TYPE T_Ctrl_SIf_DPJ_Out :
STRUCT
	///switch valve retract
	bolRetract: T_Ctrl_IoBool;
	///switch valve extend
	bolExtend: T_Ctrl_IoBool;
END_STRUCT
END_TYPE

(* stored: Version 1.1.0.1, ProductVersion 3.1.0.19
   DUT T_Ctrl_SIf_DPJ_Out: Id {5cd87c13-4e75-4d9a-81de-5ce85bf7a11a} *)
